(* CODESYS project MC500.project
   Title: MC500
   CompiledLibraryCompatibilityVersion: LeadSysStudio V3.5 SP15 Patch 4

Project tree, tasks and I/O mapping:
  Device : MC508, Leadshine Technology Co., Ltd., order no. 508101, version 3.5.15.40
      settings: RetainMode = 0; RetainStartAddr = 20480; RetainEndAddr = 524287; RetainSize = 524288; LMMVersion = 0
    application Application
      libraries: Standard, * (System); LS_IpoLib, 3.0.0.0 (Leadshine Technology Co.Ltd); LS_UtilsLib, 1.0.0.7 (Leadshine Technology Co.Ltd)
      task MainTask (cyclic, interval 500 µs, priority 0) calls M
      program M [ST]: io, io_hmi_down, io_input, io_output, io_hmi_up, cf_save_check, cf_save_apply, work
      DataMain/
        data type HMIData
        data type ConfigData
        data type SaveHelperData
        data type IOData
        data type ShapeData
      global variables GVL
      Object/
        data type Button
        data type Cylinder
        data type AirBurst
        data type Problem
        data type Pump
        data type Heater
        data type Alarm
      Enum/
        data type WorkMode
        data type State
        data type ProblemType
      DataWork/
        data type WorkData
      Symbols
      global variables PersistentVars
      AllFB/
        function StateNext [ST]
        function NPBitToPos [ST]
        function block IOWord [ST]
        function ProblemCheck [ST]
    Device Diagnose
    Network Configuration
      LocalBus Config
    Resource Usage
    SoftMotion General Axis Pool
    High_Speed_IO_Module : High Speed IO, Leadshine Technology Co., Ltd., version 3.5.15.40
        unmapped channels: Genral_IO_IN, Genral_IO_Out
    LocalBus_Master_Module : LocalBus Master, Leadshine Technology Co., Ltd., version 3.5.15.40
      PM_1616_N : PM_1616_N, Leadshine Technology Co., Ltd., version 3.5.15.40
          settings: 位置号 = 0
          unmapped channels: ErrorCode, INPUT_0, OUTPUT_0
    ModbusCOM_Master_1 : ModbusCOM RS-485 Master, Leadshine Technology Co., Ltd., version 3.5.15.40
        settings: com.Baudrate = 19200
      ModbusCOM_Furnace : ModbusCOM Slave, Leadshine Technology Co., Ltd., version 3.5.15.40
          settings: channel 00.FuncCode = 3; channel 00.ResendCount = 3; channel 00.CycleTimes = 10; channel 00.ReadRegOffSet = 8192; channel 00.IOChannel = 0; channel 00.ChannelName = 'channel 00'; channel 00.ChannelNote = ''; Vendor.SlaveID = 2; Vendor.ChannelNum = 1
          unmapped channels: ErrorCode, channel 00, channel 00
      ModbusCOM_Nozzle : ModbusCOM Slave, Leadshine Technology Co., Ltd., version 3.5.15.40
          settings: channel 00.FuncCode = 3; channel 00.ResendCount = 3; channel 00.CycleTimes = 10; channel 00.ReadRegOffSet = 8192; channel 00.IOChannel = 0; channel 00.ChannelName = 'channel 00'; channel 00.ChannelNote = ''; Vendor.ChannelNum = 1
          unmapped channels: ErrorCode, channel 00, channel 00
*)

// Device/Application/DataMain/HMIData
{ attribute 'pack_mode' := ''}
TYPE HMIData :
STRUCT
	//
	cf: ConfigData;
	cfsh: SaveHelperData;
	//
	run: BOOL;
	stop: BOOL;
	problem_fix: ARRAY[0..GVL.c_problem_i_max] OF BOOL;
	test_output: ARRAY[0..15] OF BOOL;
	test_output_sub: ARRAY[0..15] OF BOOL;
	//
	view_input: ARRAY[0..15] OF BOOL;
	view_output: ARRAY[0..15] OF BOOL;
	view_input_sub: ARRAY[0..15] OF BOOL;
	view_output_sub: ARRAY[0..15] OF BOOL;
	view_cylinder_n: ARRAY[0..GVL.c_cylinder_i_max] OF BOOL;
	view_cylinder_p: ARRAY[0..GVL.c_cylinder_i_max] OF BOOL;
	view_cylinder_lock_n: ARRAY[0..GVL.c_cylinder_i_max] OF BOOL;
	view_cylinder_lock_p: ARRAY[0..GVL.c_cylinder_i_max] OF BOOL;
	view_cylinder_pos: ARRAY[0..GVL.c_cylinder_i_max] OF INT;
	view_heater_error: ARRAY[0..GVL.c_heater_i_max] OF INT;
	view_heater_temp_c: ARRAY[0..GVL.c_heater_i_max] OF INT;
	view_heater_on: ARRAY[0..GVL.c_heater_i_max] OF BOOL;
	//
	view_mode: INT;
	view_eject_door_cycle: UDINT;
	//
	view_problem_exist: BOOL;
	view_problem_index: INT;
	view_cycle_count: UDINT;
	view_cycle_time_msec: UDINT;
	//
	view_state: ARRAY[0..7] OF INT;
	view_cpu_load: ARRAY[0..2] OF DINT;
END_STRUCT
END_TYPE

// Device/Application/DataMain/ConfigData
{ attribute 'pack_mode' := ''}
TYPE ConfigData :
STRUCT
	set_done: BOOL;
	///////////
	//MACHINE//
	///////////
	cylinder_delay_n_msec: ARRAY[0..GVL.c_cylinder_i_max] OF UINT;
	cylinder_delay_p_msec: ARRAY[0..GVL.c_cylinder_i_max] OF UINT;
	cylinder_delay_o_msec: ARRAY[0..GVL.c_cylinder_i_max] OF UINT;
	air_burst_delay_msec: ARRAY[0..GVL.c_air_burst_i_max] OF UINT;
	//
	heater_temp_target_c: ARRAY[0..GVL.c_heater_i_max] OF UINT;
	heater_tolerance_c: ARRAY[0..GVL.c_heater_i_max] OF UINT;
	heater_delay_msec: ARRAY[0..GVL.c_heater_i_max] OF UINT;
	eject_count: UINT;
END_STRUCT
END_TYPE

// Device/Application/DataMain/SaveHelperData
TYPE SaveHelperData :
STRUCT
	accept: BOOL;
	decline: BOOL;
	need_check: BOOL;
	need: BOOL;
END_STRUCT
END_TYPE

// Device/Application/DataMain/IOData
TYPE IOData :
STRUCT
	state: State;
	///////
	//MAP//
	///////
	_i: ARRAY[0..15] OF BOOL; _i_fb: IOWord;
	_i_sub: ARRAY[0..15] OF BOOL; _i_sub_fb: IOWord;
	_o: ARRAY[0..15] OF BOOL; _o_fb: IOWord;
	_o_sub: ARRAY[0..15] OF BOOL; _o_sub_fb: IOWord;
	//////
	//IN//
	//////
	i_run: Button;
	i_stop: Button;
	i_door: Button;
	//
	i_mode: WorkMode;
	i_pump: Button;
	i_die: Button;
	i_die_rotate: Button;
	i_core: Button;
	i_load: Button;
	i_eject: Button;
	i_eject_blade: Button;
	i_spray: Button;
	i_eject_door: INT;
	///////
	//OUT//
	///////
	o_pump: Pump;
	o_die: Cylinder;
	o_die_rotate: Cylinder;
	o_core: Cylinder;
	o_load: Cylinder;
	o_eject: Cylinder;
	o_eject_blade: Cylinder;
	o_spray: AirBurst;
	o_furnace: Heater;
	o_nozzle: Heater;
	o_alarm: Alarm;
	//
	eject_door_last: INT;
	eject_door_cycle: UDINT;
	mode_last: WorkMode;
	//
	problem: ARRAY[0..GVL.c_problem_i_max] OF Problem;
	problem_exist: BOOL;
	problem_index: INT; // first found problem in the list
END_STRUCT
END_TYPE

// Device/Application/DataMain/ShapeData
TYPE ShapeData :
STRUCT
	id: INT; // index, value = 0 to disable
	x: DINT; // μm
	y: DINT; // μm
	//
	va: UDINT; // μm
	vb: UDINT; // μm
	vc: UDINT; // μm
	vd: UDINT; // μm
	ve: UDINT; // μm
END_STRUCT
END_TYPE

// Device/Application/Object/Button
{ attribute 'pack_mode' := ''}
TYPE Button :
STRUCT
	on: BOOL;
	rise: R_TRIG;
	rise_physical: R_TRIG;
	fall: F_TRIG;
	fall_physical: F_TRIG;
	timer: TON;
	pos: INT;
END_STRUCT
END_TYPE

// Device/Application/Object/Cylinder
{ attribute 'pack_mode' := ''}
TYPE Cylinder :
STRUCT
	pos: INT;
	lock_n: BOOL;
	lock_p: BOOL;
	n_timer: TON;
	p_timer: TON;
	o_timer: TON;
	on_n: BOOL;
	on_p: BOOL;
	on_n_ref: POINTER TO BOOL;
	on_p_ref: POINTER TO BOOL;
END_STRUCT
END_TYPE

// Device/Application/Object/AirBurst
TYPE AirBurst :
STRUCT
	on: BOOL;
	timer: TON;
	on_ref: POINTER TO BOOL;
END_STRUCT
END_TYPE

// Device/Application/Object/Problem
TYPE Problem :
STRUCT
	on: BOOL;
	timer: TON;
	rise: R_TRIG;
	fix_rise: R_TRIG;
END_STRUCT
END_TYPE

// Device/Application/Object/Pump
TYPE Pump :
STRUCT
	on: BOOL;
	on_ref: POINTER TO BOOL;
END_STRUCT
END_TYPE

// Device/Application/Enum/WorkMode
{attribute 'qualified_only'}
{attribute 'strict'}
TYPE WorkMode :
(
	NONE   := 0,
	MANUAL := 1,
	ONCE   := 2,
	AUTO   := 3
);
END_TYPE

// Device/Application/Enum/State
{attribute 'qualified_only'}
{attribute 'strict'}
TYPE State :
(
	NONE  := 0,
	RST   := 1,
	READY := 100,
	RUN   := 101,
	DONE  := 170
);
END_TYPE

// Device/Application/Enum/ProblemType
{attribute 'qualified_only'}
{attribute 'strict'}
TYPE ProblemType :
(
	NOZZLE_UNDER_HEAT  := 0,
	FURNACE_UNDER_HEAT := 1,
	EJECT_STUCK        := 2,
	PRODUCT_STUCK      := 3
);
END_TYPE

// Device/Application/DataWork/WorkData
{ attribute 'pack_mode' := ''}
TYPE WorkData :
STRUCT
	state: INT;
	state_jump: INT;
	//
	mode: WorkMode;
	step_next: BOOL;
	eject_door_cycle: UDINT;
	//
	eject_count: UINT;
	eject_count_remain: UINT;
	eject_b_count: UINT;
	cylinder: POINTER TO Cylinder;
	//
	cycle_start_msec: ULINT;
	cycle_time_msec: UDINT;
END_STRUCT
END_TYPE

// Device/Application/Object/Heater
TYPE Heater :
STRUCT
	on: BOOL;
	error: POINTER TO INT; // error code
	temp_c: POINTER TO INT; // temperature
	temp_target_c: INT;
	tolerance_c: INT; // error when temp < (temp_target - tolerance)
	on_ref: POINTER TO BOOL;
	timer: TON;
END_STRUCT
END_TYPE

// Device/Application/Object/Alarm
TYPE Alarm :
STRUCT
	on: BOOL;
	on_ref: POINTER TO BOOL;
END_STRUCT
END_TYPE

// Device/Application/GVL
{attribute 'qualified_only'}
VAR_GLOBAL CONSTANT
	c_problem_i_max: INT := 8 - 1;
	//
	c_cylinder_i_max: INT := 6 - 1;
	c_air_burst_i_max: INT := 1 - 1;
	c_heater_i_max: INT := 2 - 1;
END_VAR

// Device/Application/PersistentVars
{attribute 'qualified_only'}
VAR_GLOBAL PERSISTENT RETAIN
END_VAR
VAR_GLOBAL PERSISTENT
	M.cf: ConfigData;
END_VAR

// Device/Application/M
PROGRAM M
VAR
	time_msec_last: ULINT;
	time_msec : ULINT;
	time_delta_sec: LREAL;
	//
	_state: INT;
	iod: IOData;
	workd: WorkData;
	hmi: HMIData;
	cfsb: Button; // config save button
	//
	i: INT;
	j: INT;
	k: INT;
	cylinders: ARRAY[0..GVL.c_cylinder_i_max] OF POINTER TO Cylinder;
	air_bursts: ARRAY[0..GVL.c_air_burst_i_max] OF POINTER TO AirBurst;
	heaters: ARRAY[0..GVL.c_heater_i_max] OF POINTER TO Heater;
END_VAR

VAR RETAIN
	cycle_count: UDINT;
	cycle_count_reset_time_msec: ULINT;
END_VAR

VAR PERSISTENT
	cf: ConfigData;
END_VAR

MC_SysLib.SysTimeRtc.SysTimeRtcHighResGet(pTimestamp:= time_msec);
time_delta_sec := ULINT_TO_LREAL(time_msec - time_msec_last) * 1E-3;
time_msec_last := time_msec;
hmi.view_state[0] := _state;
hmi.view_cpu_load[0] := load_allcore;
hmi.view_cpu_load[1] := load_core0;
hmi.view_cpu_load[2] := load_core1;
CASE _state OF
	State.NONE: // khi khởi động thì state_main = 0 tức là = State.NONE
		iod._i_fb.value := ADR(%IW0); iod._i_fb.ref := ADR(iod._i);
		iod._o_fb.value := ADR(%QW0); iod._o_fb.ref := ADR(iod._o);
		iod._i_sub_fb.value := ADR(%IW2); iod._i_sub_fb.ref := ADR(iod._i_sub);
		iod._o_sub_fb.value := ADR(%QW1); iod._o_sub_fb.ref := ADR(iod._o_sub);
		iod.o_nozzle.error := ADR(%IW3);
		iod.o_nozzle.temp_c := ADR(%IW4);
		iod.o_furnace.error := ADR(%IW6);
		iod.o_furnace.temp_c := ADR(%IW7);
		//
		iod.o_pump.on_ref          := ADR(iod._o[0]);
		iod.o_die.on_p_ref         := ADR(iod._o[1]);
		iod.o_die.on_n_ref         := ADR(iod._o[2]);
		iod.o_die_rotate.on_p_ref  := ADR(iod._o[3]);
		iod.o_die_rotate.on_n_ref  := ADR(iod._o[4]);
		iod.o_core.on_p_ref        := ADR(iod._o[5]);
		iod.o_core.on_n_ref        := ADR(iod._o[6]);
		iod.o_load.on_p_ref        := ADR(iod._o[7]);
		iod.o_load.on_n_ref        := ADR(iod._o[8]);
		iod.o_eject.on_p_ref       := ADR(iod._o[9]);
		iod.o_eject.on_n_ref       := ADR(iod._o[10]);
		iod.o_eject_blade.on_p_ref := ADR(iod._o[11]);
		iod.o_spray.on_ref         := ADR(iod._o[12]);
		iod.o_furnace.on_ref       := ADR(iod._o[13]);
		iod.o_alarm.on_ref         := ADR(iod._o[14]);
		iod.o_nozzle.on_ref        := ADR(iod._o[15]);
		//
		cylinders[0] := ADR(iod.o_die);
		cylinders[1] := ADR(iod.o_die_rotate);
		cylinders[2] := ADR(iod.o_core);
		cylinders[3] := ADR(iod.o_load);
		cylinders[4] := ADR(iod.o_eject);
		cylinders[5] := ADR(iod.o_eject_blade);
		//
		air_bursts[0] := ADR(iod.o_spray);
		//
		heaters[0] := ADR(iod.o_nozzle);
		heaters[1] := ADR(iod.o_furnace);
		//
		StateNext(_state); // chuyển tới trạng thái tiếp theo
	1:
		IF NOT cf.set_done THEN
			cf.set_done := TRUE;
		END_IF
		StateNext(_state);
	2:
		cf_save_apply();
		StateNext(_state);
	3:
		iod.state := State.RST;
		workd.state := State.RST; // reset work
		_state := State.READY; // bước vào giai đoạn chạy
	State.READY:
		io(); // kiểm tra io (gồm PLC io và HMI)
		work();
END_CASE

ACTION io:
CASE iod.state OF
	State.RST:
		iod.i_run.timer.PT := INT_TO_TIME(1_000);
		iod.mode_last := WorkMode.NONE;
		iod.i_mode := WorkMode.NONE;
		iod.state := State.READY;
	State.READY:
		io_hmi_down();
		io_input();
		io_output();
		io_hmi_up();
END_CASE
END_ACTION

ACTION io_hmi_down:
////////
//WORK//
////////
// basis
iod.i_run.rise(CLK:= hmi.run, Q=> );
iod.i_stop.rise(CLK:= hmi.stop, Q=> );
// machine
// fix problem
FOR i := 0 TO GVL.c_problem_i_max DO
	iod.problem[i].fix_rise(CLK:= hmi.problem_fix[i], Q=> );
END_FOR
//////////////
//SAVE BASIC//
//////////////
IF hmi.cfsh.need_check THEN
	cf_save_check();
	hmi.cfsh.need_check := FALSE;
END_IF
cfsb.rise(CLK:= hmi.cfsh.accept, Q=> ); // Trên HMI sẽ xuất hiện nút save khi biến hmi_data.save_need = true.
IF cfsb.rise.Q THEN
	cf := hmi.cf;
	cf_save_apply();
	hmi.cfsh.need := FALSE;
	hmi.cfsh.accept := FALSE;
	hmi.cfsh.decline := FALSE;
END_IF
cfsb.rise_physical(CLK:= hmi.cfsh.decline, Q=> );
IF cfsb.rise_physical.Q THEN
	hmi.cf := cf;
	hmi.cfsh.need := FALSE;
	hmi.cfsh.accept := FALSE;
	hmi.cfsh.decline := FALSE;
END_IF
END_ACTION

ACTION io_input:
//////////////////
//PHYSICAL INPUT//
//////////////////
iod._i_fb(control:= 1);
iod._o_fb(control:= 1);
iod._i_sub_fb(control:= 1);
iod._o_sub_fb(control:= 1);
//
iod.i_run.rise_physical(CLK:= iod._i[14], Q=> );
iod.i_stop.fall_physical(CLK:= iod._i[15], Q=> );
iod.i_door.fall_physical(CLK:= iod._i[0], Q=> );
//
iod.i_eject_door := NPBitToPos(n:= iod._i[1], p:= iod._i[2]);
IF iod.i_eject_door <> 0 AND iod.i_eject_door <> iod.eject_door_last THEN
	IF iod.i_eject_door = 1 THEN
		iod.eject_door_cycle := iod.eject_door_cycle + 1;
	END_IF
	iod.eject_door_last := iod.i_eject_door;
END_IF
i := BOOL_TO_INT(iod._i_sub[0]) + BOOL_TO_INT(iod._i_sub[1]) * 2 + BOOL_TO_INT(iod._i_sub[2]) * 4;
CASE i OF
    3: iod.i_mode := WorkMode.MANUAL;
	0: iod.i_mode := WorkMode.ONCE;
	6: iod.i_mode := WorkMode.AUTO;
	ELSE iod.i_mode := WorkMode.NONE;
END_CASE
iod.i_pump.on         := iod._i_sub[3];
iod.i_die.pos         := NPBitToPos(n:= iod._i_sub[5], p:= iod._i_sub[4]);
iod.i_die_rotate.pos  := NPBitToPos(n:= iod._i_sub[7], p:= iod._i_sub[6]);
iod.i_core.pos        := NPBitToPos(n:= iod._i_sub[9], p:= iod._i_sub[8]);
iod.i_load.pos        := NPBitToPos(n:= iod._i_sub[11], p:= iod._i_sub[10]);
iod.i_eject.pos       := NPBitToPos(n:= iod._i_sub[13], p:= iod._i_sub[12]);
iod.i_eject_blade.pos := NPBitToPos(n:= FALSE, p:= iod._i_sub[14]);
iod.i_spray.on        := iod._i_sub[15];
////////////
//CYLINDER//
////////////
// n, p
iod.o_die.n_timer(IN:= iod.o_die.on_n AND iod._i[5], PT:= , Q=> , ET=> );
iod.o_die.p_timer(IN:= iod.o_die.on_p AND iod._i[3] AND iod._i[4], PT:= , Q=> , ET=> );
iod.o_core.n_timer(IN:= iod.o_core.on_n AND iod._i[7], PT:= , Q=> , ET=> );
iod.o_core.p_timer(IN:= iod.o_core.on_p AND iod._i[6], PT:= , Q=> , ET=> );
iod.o_load.n_timer(IN:= iod.o_load.on_n AND iod._i[8], PT:= , Q=> , ET=> );
iod.o_load.p_timer(IN:= iod.o_load.on_p, PT:= , Q=> , ET=> );
iod.o_eject.n_timer(IN:= iod.o_eject.on_n AND iod._i[10], PT:= , Q=> , ET=> );
iod.o_eject.p_timer(IN:= iod.o_eject.on_p AND iod._i[9], PT:= , Q=> , ET=> );
iod.o_eject_blade.n_timer(IN:= NOT iod.o_eject_blade.on_p AND iod._i[11], PT:= , Q=> , ET=> );
iod.o_eject_blade.p_timer(IN:= iod.o_eject_blade.on_p, PT:= , Q=> , ET=> );
// o
iod.o_die.o_timer(IN:= iod.o_die.pos <> 0, PT:= , Q=> , ET=> );
iod.o_core.o_timer(IN:= iod.o_core.pos <> 0, PT:= , Q=> , ET=> );
iod.o_load.o_timer(IN:= iod.o_load.pos <> 0, PT:= , Q=> , ET=> );
iod.o_eject.o_timer(IN:= iod.o_eject.pos <> 0, PT:= , Q=> , ET=> );
// lock n, p
iod.o_die.lock_n         := NOT (iod.o_load.n_timer.Q);
iod.o_die.lock_p         := NOT (iod.o_eject.n_timer.Q AND iod.o_eject_blade.n_timer.Q);
iod.o_die_rotate.lock_n  := NOT (iod.i_mode = WorkMode.MANUAL AND iod.i_run.rise_physical.CLK);
iod.o_die_rotate.lock_p  := iod.o_die_rotate.lock_n;
iod.o_core.lock_n        := NOT (iod.o_load.n_timer.Q AND iod.o_eject_blade.n_timer.Q);
iod.o_core.lock_p        := FALSE;
iod.o_load.lock_n        := FALSE;
iod.o_load.lock_p        := NOT (iod.o_die.p_timer.Q AND iod.o_core.p_timer.Q AND NOT iod.o_core.o_timer.Q);
iod.o_eject.lock_n       := FALSE;
iod.o_eject.lock_p       := NOT iod.o_die.n_timer.Q;
iod.o_eject_blade.lock_n := FALSE;
iod.o_eject_blade.lock_p := NOT (iod.o_die.n_timer.Q AND iod.o_core.p_timer.Q);
///////////
//PROBLEM//
///////////
// exist
FOR i := 0 TO GVL.c_problem_i_max DO
	iod.problem[i].rise(CLK:= iod.problem[i].on, Q=> );
END_FOR
ProblemCheck(ref:= ADR(iod.problem), exist=> iod.problem_exist, index=> iod.problem_index);
iod.o_alarm.on := iod.problem_exist;
// fix
IF iod.problem[ProblemType.NOZZLE_UNDER_HEAT].fix_rise.Q THEN
	iod.problem[ProblemType.NOZZLE_UNDER_HEAT].on := FALSE;
	hmi.problem_fix[ProblemType.NOZZLE_UNDER_HEAT] := FALSE;
END_IF
IF iod.problem[ProblemType.FURNACE_UNDER_HEAT].fix_rise.Q THEN
	iod.problem[ProblemType.FURNACE_UNDER_HEAT].on := FALSE;
	hmi.problem_fix[ProblemType.FURNACE_UNDER_HEAT] := FALSE;
END_IF
IF iod.problem[ProblemType.EJECT_STUCK].fix_rise.Q THEN
	iod.problem[ProblemType.EJECT_STUCK].on := FALSE;
	hmi.problem_fix[ProblemType.EJECT_STUCK] := FALSE;
END_IF
IF iod.problem[ProblemType.PRODUCT_STUCK].fix_rise.Q THEN
	iod.problem[ProblemType.PRODUCT_STUCK].on := FALSE;
	hmi.problem_fix[ProblemType.PRODUCT_STUCK] := FALSE;
END_IF
///////////////////
//MACHINE PROCESS//
///////////////////
// mode change
IF iod.i_mode <> iod.mode_last THEN
	IF (workd.state = State.READY AND iod.i_mode = WorkMode.MANUAL AND
		iod.i_pump.on AND
		iod.i_die.pos = 0 AND
		iod.i_die_rotate.pos = 0 AND
		iod.i_core.pos = 0 AND
		iod.i_load.pos = 0 AND
		iod.i_eject.pos = 0 AND
		iod.i_eject_blade.pos = 0 AND
		NOT iod.i_spray.on
	) THEN
		workd.mode := WorkMode.MANUAL;
	END_IF
	IF (workd.mode = WorkMode.MANUAL AND
		workd.state = State.READY AND iod.i_mode = WorkMode.ONCE AND
		iod.o_pump.on AND
		iod.o_die.n_timer.Q AND
		iod.o_die_rotate.pos = 0 AND
		iod.o_core.p_timer.Q AND
		iod.o_load.n_timer.Q AND
		iod.o_eject.n_timer.Q AND
		iod.o_eject_blade.n_timer.Q AND
		NOT iod.o_spray.on
	) THEN
		workd.mode := WorkMode.ONCE;
	END_IF
	IF workd.mode = WorkMode.ONCE AND iod.i_mode = WorkMode.AUTO THEN
		workd.mode := WorkMode.AUTO;
	END_IF
	IF workd.mode = WorkMode.AUTO AND iod.i_mode = WorkMode.ONCE THEN
		workd.mode := WorkMode.ONCE;
	END_IF
	iod.mode_last := iod.i_mode;
END_IF
IF workd.state = State.READY AND workd.mode = WorkMode.MANUAL THEN
	iod.o_pump.on         := iod.i_pump.on;
	iod.o_die.pos         := iod.i_die.pos;
	iod.o_die_rotate.pos  := iod.i_die_rotate.pos;
	iod.o_core.pos        := iod.i_core.pos;
	iod.o_load.pos        := iod.i_load.pos;
	iod.o_eject.pos       := iod.i_eject.pos;
	iod.o_eject_blade.pos := iod.i_eject_blade.pos;
	iod.o_spray.on        := iod.i_spray.on;
END_IF
// run
IF iod.i_run.rise.Q OR iod.i_run.rise_physical.Q THEN
	workd.step_next := TRUE;
	IF (iod.i_stop.fall_physical.CLK AND
		(workd.state = State.READY OR workd.state = State.DONE) AND
		(workd.mode = WorkMode.ONCE OR workd.mode = WorkMode.AUTO)
	) THEN
		workd.state := State.RUN;
	END_IF
END_IF
IF workd.mode = WorkMode.AUTO THEN
	workd.step_next := TRUE;
	IF workd.state = State.DONE THEN
		workd.state := State.RUN;
	END_IF
END_IF
// stop
IF iod.i_stop.rise.Q OR iod.i_stop.fall_physical.Q OR iod.i_door.fall_physical.Q THEN
	CASE workd.mode OF
		WorkMode.MANUAL:
			workd.state := State.RST;
			workd.mode := WorkMode.NONE;
		WorkMode.ONCE:
			workd.step_next := FALSE;
			workd.mode := WorkMode.MANUAL;
		WorkMode.AUTO:
			workd.step_next := FALSE;
			workd.mode := WorkMode.ONCE;
	END_CASE
END_IF
END_ACTION

ACTION io_output:
/////////////
//AIR BURST//
/////////////
FOR i := 0 TO GVL.c_air_burst_i_max DO
	air_bursts[i]^.timer(IN:= air_bursts[i]^.on, PT:= , Q=> , ET=> );
	IF air_bursts[i]^.timer.Q THEN
		air_bursts[i]^.on := FALSE;
	END_IF
END_FOR
//////////
//HEATER//
//////////
FOR i := 0 TO GVL.c_heater_i_max DO
	heaters[i]^.timer(IN:= , PT:= , Q=> , ET=> );
	IF heaters[i]^.error^ = 0 THEN
		IF heaters[i]^.temp_c^ < heaters[i]^.temp_target_c THEN
			heaters[i]^.timer.IN := TRUE;
			IF heaters[i]^.timer.Q THEN
				heaters[i]^.on := TRUE;
			END_IF
		ELSE
			heaters[i]^.timer.IN := FALSE;
			heaters[i]^.on := FALSE;
		END_IF
	ELSE
		heaters[i]^.timer.IN := FALSE;
		heaters[i]^.on := FALSE;
	END_IF
END_FOR
////////////
//PHYSICAL//
////////////
iod.o_die.on_n         := iod.o_die.pos         < 0 AND NOT iod.o_die.lock_n;
iod.o_die.on_p         := iod.o_die.pos         > 0 AND NOT iod.o_die.lock_p;
iod.o_core.on_n        := iod.o_core.pos        < 0 AND NOT iod.o_core.lock_n;
iod.o_core.on_p        := iod.o_core.pos        > 0 AND NOT iod.o_core.lock_p;
iod.o_load.on_n        := iod.o_load.pos        < 0 AND NOT iod.o_load.lock_n;
iod.o_load.on_p        := iod.o_load.pos        > 0 AND NOT iod.o_load.lock_p;
iod.o_eject.on_n       := iod.o_eject.pos       < 0 AND NOT iod.o_eject.lock_n;
iod.o_eject.on_p       := iod.o_eject.pos       > 0 AND NOT iod.o_eject.lock_p;
iod.o_eject_blade.on_p := iod.o_eject_blade.pos > 0 AND NOT iod.o_eject_blade.lock_p;
iod.o_die_rotate.on_n  := iod.o_die_rotate.pos  < 0 AND NOT iod.o_die_rotate.lock_n;
iod.o_die_rotate.on_p  := iod.o_die_rotate.pos  > 0 AND NOT iod.o_die_rotate.lock_p;
//
iod.o_die.on_n_ref^         := iod.o_die.on_n   AND NOT iod.o_die.o_timer.Q;
iod.o_die.on_p_ref^         := iod.o_die.on_p   AND NOT iod.o_die.o_timer.Q;
iod.o_core.on_n_ref^        := iod.o_core.on_n  AND NOT iod.o_core.o_timer.Q;
iod.o_core.on_p_ref^        := iod.o_core.on_p  AND NOT iod.o_core.o_timer.Q;
iod.o_load.on_n_ref^        := iod.o_load.on_n  AND NOT iod.o_load.o_timer.Q;
iod.o_load.on_p_ref^        := iod.o_load.on_p  AND NOT iod.o_load.o_timer.Q;
iod.o_eject.on_n_ref^       := iod.o_eject.on_n AND NOT iod.o_eject.o_timer.Q;
iod.o_eject.on_p_ref^       := iod.o_eject.on_p AND NOT iod.o_eject.o_timer.Q;
iod.o_eject_blade.on_p_ref^ := iod.o_eject_blade.on_p;
iod.o_die_rotate.on_n_ref^  := iod.o_die_rotate.on_n;
iod.o_die_rotate.on_p_ref^  := iod.o_die_rotate.on_p;
iod.o_pump.on_ref^          := iod.o_pump.on;
iod.o_spray.on_ref^         := iod.o_spray.on;
iod.o_furnace.on_ref^       := iod.o_furnace.on;
iod.o_nozzle.on_ref^        := iod.o_nozzle.on;
iod.o_alarm.on_ref^        := iod.o_alarm.on;
//
iod._o_fb(control:= 2);
iod._o_sub_fb(control:= 2);
END_ACTION

ACTION io_hmi_up:
/////////
//STATE//
/////////
hmi.view_state[1] := workd.state;
///////////////
//PHYSICAL IO//
///////////////
FOR i := 0 TO 15 BY 1 DO
	hmi.view_input[i] := iod._i[i];
	hmi.view_output[i] := iod._o[i];
	hmi.view_input_sub[i] := iod._i_sub[i];
	hmi.view_output_sub[i] := iod._o_sub[i];
END_FOR
/////////////////
//MACHINE STATE//
/////////////////
hmi.view_problem_exist := iod.problem_exist;
hmi.view_problem_index := iod.problem_index;
///////////
//MACHINE//
///////////
FOR i := 0 TO GVL.c_cylinder_i_max BY 1 DO
	hmi.view_cylinder_n[i] := cylinders[i]^.n_timer.Q;
	hmi.view_cylinder_p[i] := cylinders[i]^.p_timer.Q;
	hmi.view_cylinder_lock_n[i] := cylinders[i]^.lock_n;
	hmi.view_cylinder_lock_p[i] := cylinders[i]^.lock_p;
	hmi.view_cylinder_pos[i] := cylinders[i]^.pos;
END_FOR
FOR i := 0 TO GVL.c_heater_i_max BY 1 DO
	hmi.view_heater_error[i] := heaters[i]^.error^;
	hmi.view_heater_temp_c[i] := heaters[i]^.temp_c^;
	hmi.view_heater_on[i] := heaters[i]^.on;
END_FOR
hmi.view_mode := workd.mode;
hmi.view_eject_door_cycle := iod.eject_door_cycle;
/////////
//OTHER//
/////////
hmi.view_cycle_count := cycle_count;
hmi.view_cycle_time_msec := workd.cycle_time_msec;
END_ACTION

ACTION cf_save_check:
hmi.cfsh.need := (
	cf.eject_count <> hmi.cf.eject_count
);
FOR i := 0 TO GVL.c_cylinder_i_max BY 1 DO
	hmi.cfsh.need := (hmi.cfsh.need OR
		cf.cylinder_delay_n_msec[i] <> hmi.cf.cylinder_delay_n_msec[i] OR
		cf.cylinder_delay_p_msec[i] <> hmi.cf.cylinder_delay_p_msec[i] OR
		cf.cylinder_delay_o_msec[i] <> hmi.cf.cylinder_delay_o_msec[i]
	);
END_FOR
FOR i := 0 TO GVL.c_air_burst_i_max BY 1 DO
	hmi.cfsh.need := (hmi.cfsh.need OR
		cf.air_burst_delay_msec[i] <> hmi.cf.air_burst_delay_msec[i]
	);
END_FOR
FOR i := 0 TO GVL.c_heater_i_max BY 1 DO
	hmi.cfsh.need := (hmi.cfsh.need OR
		cf.heater_temp_target_c[i] <> hmi.cf.heater_temp_target_c[i] OR
		cf.heater_tolerance_c[i] <> hmi.cf.heater_tolerance_c[i] OR
		cf.heater_delay_msec[i] <> hmi.cf.heater_delay_msec[i]
	);
END_FOR
END_ACTION

ACTION cf_save_apply:
/////////////
//LIMIT AIR//
/////////////
FOR i := 0 TO GVL.c_cylinder_i_max DO
	cf.cylinder_delay_n_msec[i] := MAX(0_100, MIN(9_000, cf.cylinder_delay_n_msec[i]));
	cf.cylinder_delay_p_msec[i] := MAX(0_100, MIN(9_000, cf.cylinder_delay_p_msec[i]));
	cf.cylinder_delay_o_msec[i] := MAX(3_000, MIN(60_000, cf.cylinder_delay_o_msec[i]));
END_FOR
FOR i := 0 TO GVL.c_air_burst_i_max DO
	cf.air_burst_delay_msec[i] := MAX(0_100, MIN(9_000, cf.air_burst_delay_msec[i]));
END_FOR
/////////////
//APPLY AIR//
/////////////
FOR i := 0 TO GVL.c_cylinder_i_max DO
	cylinders[i]^.n_timer.PT := UINT_TO_TIME(cf.cylinder_delay_n_msec[i]);
	cylinders[i]^.p_timer.PT := UINT_TO_TIME(cf.cylinder_delay_p_msec[i]);
	cylinders[i]^.o_timer.PT := UINT_TO_TIME(cf.cylinder_delay_o_msec[i]);
END_FOR
FOR i := 0 TO GVL.c_air_burst_i_max DO
	air_bursts[i]^.timer.PT := UINT_TO_TIME(cf.air_burst_delay_msec[i]);
END_FOR
/////////////////
//LIMIT MACHINE//
/////////////////
FOR i := 0 TO GVL.c_heater_i_max DO
	cf.heater_temp_target_c[i] := MAX(10, MIN(900, cf.heater_temp_target_c[i]));
	cf.heater_tolerance_c[i] := MAX(1, MIN(50, cf.heater_tolerance_c[i]));
	cf.heater_delay_msec[i] := MAX(3_000, MIN(60_000, cf.heater_delay_msec[i]));
END_FOR
cf.eject_count := MAX(1, MIN(5, cf.eject_count));
/////////////////
//APPLY MACHINE//
/////////////////
FOR i := 0 TO GVL.c_heater_i_max DO
	heaters[i]^.temp_target_c := UINT_TO_INT(cf.heater_temp_target_c[i]);
	heaters[i]^.tolerance_c := UINT_TO_INT(cf.heater_tolerance_c[i]);
	heaters[i]^.timer.PT := UINT_TO_TIME(cf.heater_delay_msec[i]);
END_FOR
workd.eject_count := cf.eject_count;
/////////
//FINAL//
/////////
hmi.cf := cf;
END_ACTION

ACTION work:
CASE workd.state OF
	State.RST:
		StateNext(workd.state);
	2: // load ↑
		workd.cylinder := ADR(iod.o_load);
		workd.cylinder^.pos := 0;
		StateNext(workd.state);
	3:
		IF NOT workd.cylinder^.o_timer.Q THEN
			workd.cylinder^.pos := -1;
			StateNext(workd.state);
		END_IF
	4:
		IF workd.cylinder^.n_timer.Q THEN
			StateNext(workd.state);
		END_IF
	5: // eject blade ↑
		workd.cylinder := ADR(iod.o_eject_blade);
		workd.cylinder^.pos := 0;
		StateNext(workd.state);
	6:
		IF NOT workd.cylinder^.o_timer.Q THEN
			workd.cylinder^.pos := -1;
			StateNext(workd.state);
		END_IF
	7:
		IF workd.cylinder^.n_timer.Q THEN
			StateNext(workd.state);
		END_IF
	8:
		workd.state := State.READY;
	///////
	//RUN//
	///////
	State.RUN:
		IF iod.o_nozzle.temp_c^ < (iod.o_nozzle.temp_target_c - iod.o_nozzle.tolerance_c) OR iod.o_nozzle.error^ <> 0 THEN
			iod.problem[ProblemType.NOZZLE_UNDER_HEAT].on := TRUE;
		END_IF
		IF iod.o_furnace.temp_c^ < (iod.o_furnace.temp_target_c - iod.o_furnace.tolerance_c) OR iod.o_furnace.error^ <> 0 THEN
			iod.problem[ProblemType.FURNACE_UNDER_HEAT].on := TRUE;
		END_IF
		IF iod.problem[ProblemType.NOZZLE_UNDER_HEAT].on OR iod.problem[ProblemType.FURNACE_UNDER_HEAT].on THEN
			workd.state := State.READY;
		ELSE
			workd.cycle_start_msec := time_msec;
			workd.step_next := FALSE;
			StateNext(workd.state);
		END_IF
	102: // spray
		IF workd.step_next THEN
			workd.step_next := FALSE;
			iod.o_spray.on := TRUE;
			StateNext(workd.state);
		END_IF
	103:
		IF NOT iod.o_spray.on THEN
			workd.state := 121;
		END_IF
	////////
	//CAST//
	////////
	121: // die →
		IF workd.step_next THEN
			workd.step_next := FALSE;
			workd.cylinder := ADR(iod.o_die);
			workd.cylinder^.pos := 0;
			StateNext(workd.state);
		END_IF
	122:
		IF NOT workd.cylinder^.o_timer.Q THEN
			workd.cylinder^.pos := 1;
			StateNext(workd.state);
		END_IF
	123:
		IF workd.cylinder^.p_timer.Q THEN
			StateNext(workd.state);
		END_IF
	124: // core →, load ↓↑
		IF workd.step_next THEN
			workd.step_next := FALSE;
			workd.cylinder := ADR(iod.o_core);
			workd.cylinder^.pos := 0;
			StateNext(workd.state);
		END_IF
	125:
		IF NOT workd.cylinder^.o_timer.Q THEN
			workd.cylinder^.pos := 1;
			StateNext(workd.state);
		END_IF
	126:
		IF workd.cylinder^.p_timer.Q THEN
			workd.cylinder := ADR(iod.o_load);
			workd.cylinder^.pos := 0;
			StateNext(workd.state);
		END_IF
	127:
		IF NOT workd.cylinder^.o_timer.Q THEN
			workd.cylinder^.pos := 1;
			StateNext(workd.state);
		END_IF
	128:
		IF workd.cylinder^.p_timer.Q THEN
			workd.cylinder^.pos := 0;
			StateNext(workd.state);
		END_IF
	129:
		IF NOT workd.cylinder^.o_timer.Q THEN
			workd.cylinder^.pos := -1;
			StateNext(workd.state);
		END_IF
	130:
		IF workd.cylinder^.n_timer.Q THEN
			StateNext(workd.state);
		END_IF
	131: // die ←
		IF workd.step_next THEN
			workd.step_next := FALSE;
			workd.cylinder := ADR(iod.o_die);
			workd.eject_door_cycle := iod.eject_door_cycle;
			workd.cylinder^.pos := 0;
			StateNext(workd.state);
		END_IF
	132:
		IF NOT workd.cylinder^.o_timer.Q THEN
			workd.cylinder^.pos := -1;
			StateNext(workd.state);
		END_IF
	133:
		IF workd.cylinder^.n_timer.Q THEN
			workd.eject_count_remain := workd.eject_count;
			workd.state := 141;
		END_IF
	/////////
	//EJECT//
	/////////
	141: // eject → ←
		IF workd.step_next THEN
			workd.step_next := FALSE;
			workd.cylinder := ADR(iod.o_eject);
			workd.eject_count_remain := workd.eject_count_remain - 1;
			workd.cylinder^.pos := 0;
			StateNext(workd.state);
		END_IF
	142:
		IF NOT workd.cylinder^.o_timer.Q THEN
			workd.cylinder^.pos := 1;
			StateNext(workd.state);
		END_IF
	143:
		IF workd.cylinder^.o_timer.Q THEN
			iod.problem[ProblemType.EJECT_STUCK].on := TRUE;
			workd.state_jump := 141;
			workd.state := 156; // jump -> eject stuck
		ELSE
			IF workd.cylinder^.p_timer.Q THEN
				workd.cylinder^.pos := 0;
				StateNext(workd.state);
			END_IF
		END_IF
	144:
		IF NOT workd.cylinder^.o_timer.Q THEN
			workd.cylinder^.pos := -1;
			StateNext(workd.state);
		END_IF
	145:
		IF workd.cylinder^.o_timer.Q THEN
			iod.problem[ProblemType.EJECT_STUCK].on := TRUE;
			workd.state_jump := 141;
			workd.state := 156; // jump -> eject stuck
		ELSE
			IF workd.cylinder^.n_timer.Q THEN
				StateNext(workd.state);
			END_IF
		END_IF
	146:
		IF workd.eject_count_remain > 0 THEN
			workd.state := 141;
		ELSE
			workd.eject_b_count := 0;
			workd.state := 151;
		END_IF
	///////////////
	//EJECT BLADE//
	///////////////
	151: // eject blade ↓↑
		IF workd.step_next THEN
			workd.step_next := FALSE;
			workd.cylinder := ADR(iod.o_eject_blade);
			workd.cylinder^.pos := 1;
			StateNext(workd.state);
		END_IF
	152:
		IF workd.cylinder^.p_timer.Q THEN
			workd.cylinder^.pos := -1;
			StateNext(workd.state);
		END_IF
	153:
		IF workd.cylinder^.n_timer.Q THEN
			workd.eject_b_count := workd.eject_b_count + 1;
			StateNext(workd.state);
		END_IF
	154: // done || eject blade ↓↑
		IF iod.eject_door_cycle > workd.eject_door_cycle THEN
			workd.state := 161;
		ELSE
			IF workd.eject_b_count > 2 THEN
				iod.problem[ProblemType.PRODUCT_STUCK].on := TRUE;
				workd.state_jump := workd.state;
				workd.state := 157; // jump -> product stuck
			ELSE
				workd.state := 151;
			END_IF
		END_IF
	156: // eject stuck
		IF NOT iod.problem[ProblemType.EJECT_STUCK].on THEN
			workd.eject_count_remain := workd.eject_count;
			workd.state := workd.state_jump;
		END_IF
	157: // product stuck
		IF NOT iod.problem[ProblemType.PRODUCT_STUCK].on THEN
			workd.state := workd.state_jump;
		END_IF
	////////
	//DONE//
	////////
	161:
		workd.state := State.DONE;
		workd.cycle_time_msec := ULINT_TO_UDINT(time_msec - workd.cycle_start_msec);
		IF (time_msec - cycle_count_reset_time_msec) > 86400_000 THEN
			cycle_count := 0;
			cycle_count_reset_time_msec := (time_msec / 86400_000) * 86400_000;
		END_IF
		cycle_count := cycle_count + 1;
END_CASE
END_ACTION

END_PROGRAM

// Device/Application/AllFB/StateNext
FUNCTION StateNext
VAR_INPUT
	state: REFERENCE TO INT;
END_VAR
VAR
END_VAR

state := state + 1;

END_FUNCTION

// Device/Application/AllFB/NPBitToPos
FUNCTION NPBitToPos : INT
VAR_INPUT
	n: BOOL;
	p: BOOL;
END_VAR
VAR
	value: INT;
END_VAR

value := BOOL_TO_INT(n) + BOOL_TO_INT(p) * 2;
CASE value OF
	1: NPBitToPos := -1;
	2: NPBitToPos := +1;
	ELSE NPBitToPos := 0;
END_CASE

END_FUNCTION

// Device/Application/AllFB/ProblemCheck
FUNCTION ProblemCheck
VAR_INPUT
	ref: POINTER TO ARRAY[0..GVL.c_problem_i_max] OF Problem;
END_VAR
VAR_OUTPUT
	exist: BOOL;
	index: INT;
END_VAR
VAR
	i: INT;
	_exist: BOOL;
END_VAR

_exist := FALSE;
FOR i := 0 TO GVL.c_problem_i_max DO
	IF ref^[i].on THEN
		_exist := TRUE;
		index := i;
		EXIT;
	END_IF
END_FOR
exist := _exist;

END_FUNCTION

// Device/Application/AllFB/IOWord
FUNCTION_BLOCK IOWord
VAR_INPUT
	control: INT; // 1: read, 2: write
	value: POINTER TO WORD;
	ref: POINTER TO ARRAY[0..15] OF BOOL;
END_VAR
VAR
	i: INT;
	ju: UINT;
	jw: WORD;
	v: UINT;
END_VAR

CASE control OF
	1:
		FOR i := 0 TO 15 BY 1 DO
			jw := SHL(1, i); // dịch chuyển bit về bên trái, vd: 1 = 0000_0000_0000_0001 -> SHL(1, 1) = 0000_0000_0000_0010
			ref^[i] := (value^ AND jw) > 0; // phép toán bit AND, vd 0000_0000_0000_0010 AND 0100_0110_0101_0010 = 0000_0000_0000_0010 > 0
		END_FOR
	2:
		v := 0;
		FOR i := 0 TO 15 BY 1 DO
			ju := SHL(1, i);
			v := v + BOOL_TO_UINT(ref^[i]) * ju;
		END_FOR
		value^ := v;
END_CASE

END_FUNCTION_BLOCK
